% RSLogix 500 project I2A JOB 12-MITCH (NOTDONE)_BAK037.RSS, saved by version 10.00.00.00 %
PROJECT "ML01B"    % processor: Bul.1763 MicroLogix 1100 Series B %

PROGRAM FILES
  LAD 2   9 rungs

DATA FILES
  O0 OUTPUT  4 elements
  I1 INPUT  6 elements
  S2 STATUS  66 elements
  B3 BINARY  1 elements
  T4 TIMER  1 elements
  C5 COUNTER  1 elements
  R6 CONTROL  1 elements
  N7 INTEGER  1 elements
  F8 FLOAT  1 elements

LADDER 2
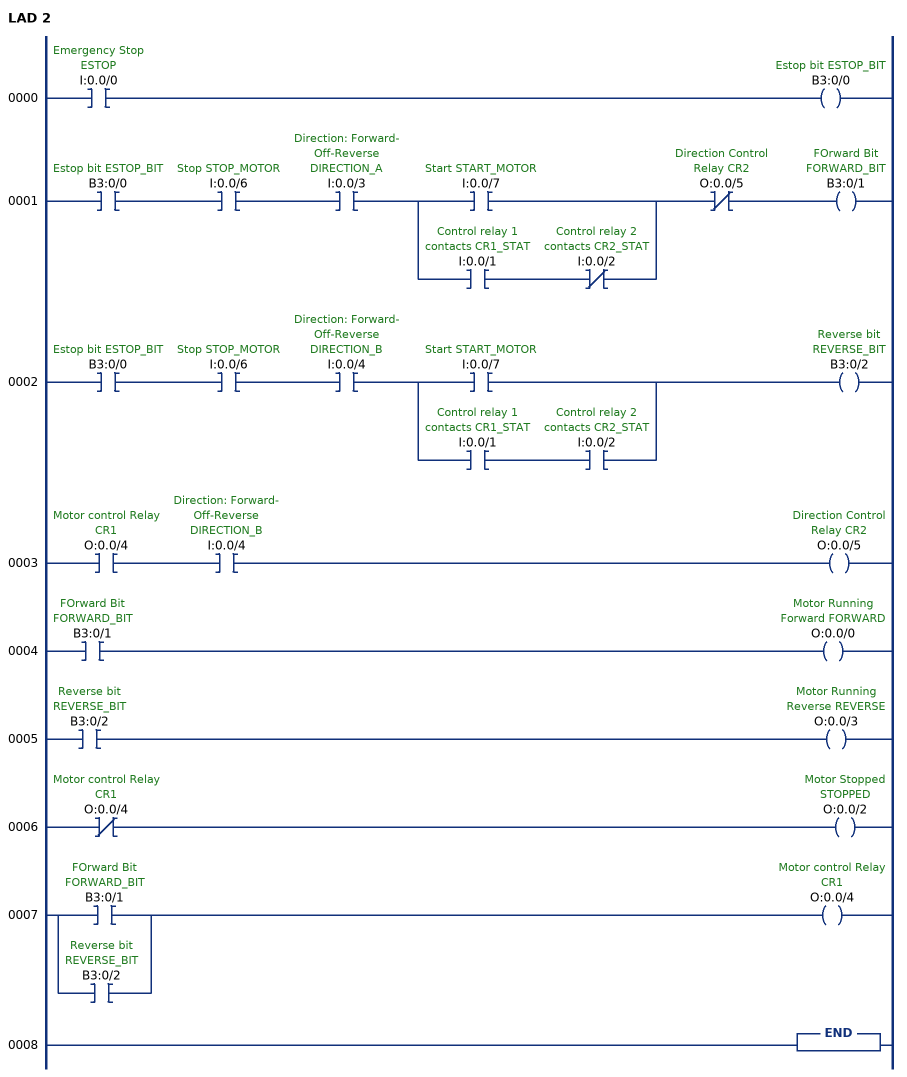
% Rung: 0 %
SOR XIC I:0.0/0 OTE B3:0/0 EOR
%   I:0.0/0  ESTOP  "Emergency Stop" %
%   B3:0/0  ESTOP_BIT  "Estop bit" %
% Rung: 1 %
SOR XIC B3:0/0 XIC I:0.0/6 XIC I:0.0/3 BST XIC I:0.0/7 NXB XIC I:0.0/1 XIO I:0.0/2 BND XIO O:0.0/5 OTE B3:0/1 EOR
%   B3:0/0  ESTOP_BIT  "Estop bit" %
%   I:0.0/6  STOP_MOTOR  "Stop" %
%   I:0.0/3  DIRECTION_A  "Direction: Forward- Off-Reverse" %
%   I:0.0/7  START_MOTOR  "Start" %
%   I:0.0/1  CR1_STAT  "Control relay 1 contacts" %
%   I:0.0/2  CR2_STAT  "Control relay 2 contacts" %
%   O:0.0/5  CR2  "Direction Control Relay" %
%   B3:0/1  FORWARD_BIT  "FOrward Bit" %
% Rung: 2 %
SOR XIC B3:0/0 XIC I:0.0/6 XIC I:0.0/4 BST XIC I:0.0/7 NXB XIC I:0.0/1 XIC I:0.0/2 BND OTE B3:0/2 EOR
%   B3:0/0  ESTOP_BIT  "Estop bit" %
%   I:0.0/6  STOP_MOTOR  "Stop" %
%   I:0.0/4  DIRECTION_B  "Direction: Forward- Off-Reverse" %
%   I:0.0/7  START_MOTOR  "Start" %
%   I:0.0/1  CR1_STAT  "Control relay 1 contacts" %
%   I:0.0/2  CR2_STAT  "Control relay 2 contacts" %
%   B3:0/2  REVERSE_BIT  "Reverse bit" %
% Rung: 3 %
SOR XIC O:0.0/4 XIC I:0.0/4 OTE O:0.0/5 EOR
%   O:0.0/4  CR1  "Motor control Relay" %
%   I:0.0/4  DIRECTION_B  "Direction: Forward- Off-Reverse" %
%   O:0.0/5  CR2  "Direction Control Relay" %
% Rung: 4 %
SOR XIC B3:0/1 OTE O:0.0/0 EOR
%   B3:0/1  FORWARD_BIT  "FOrward Bit" %
%   O:0.0/0  FORWARD  "Motor Running Forward" %
% Rung: 5 %
SOR XIC B3:0/2 OTE O:0.0/3 EOR
%   B3:0/2  REVERSE_BIT  "Reverse bit" %
%   O:0.0/3  REVERSE  "Motor Running Reverse" %
% Rung: 6 %
SOR XIO O:0.0/4 OTE O:0.0/2 EOR
%   O:0.0/4  CR1  "Motor control Relay" %
%   O:0.0/2  STOPPED  "Motor Stopped" %
% Rung: 7 %
SOR BST XIC B3:0/1 NXB XIC B3:0/2 BND OTE O:0.0/4 EOR
%   B3:0/1  FORWARD_BIT  "FOrward Bit" %
%   B3:0/2  REVERSE_BIT  "Reverse bit" %
%   O:0.0/4  CR1  "Motor control Relay" %
% Rung: 8 %
SOR END EOR

OTHER DOCUMENTED ADDRESSES
  I:0.0/5  2PSSA  "2 position selector switch A"
  I:0.0/8  PB3  "Jog"
  O:0.0/1  YELLOWLT

DATA TABLE (non-zero values as saved)
DATA B3
% B3:0 % 0X0001
